Staubli VAL3: getJointData.pgx

public program getJointData(string x_sItem (dimensions=1), num x_nIndex (dimensions=1), joint& x_jJoint (dimensions=1), bool& x_bResult (dimensions=1))
  local num i
  local num l_nResult
  local string l_sSession
begin
  // get the joint data from the specific session...
  x_bResult=false
  call saveData:getSession(l_sSession)
  // get the colletion type...
  if sSession!=l_sSession
    // copy back
    sSession=l_sSession
    // load the actual one
    l_nResult=jt:libLoad(saveData:sPathTraj+"JPOINT")
    delay(0)
  endIf
  // use the type...
  if l_nResult==0 and isDefined(jt:tTraj[x_sItem]) and size(jt:tTraj[x_sItem].tData.jJoint)>x_nIndex
    // get the JOINT DATA
    x_jJoint=jt:tTraj[x_sItem].tData.jJoint[x_nIndex]
    delay(0)
    x_bResult=true
  endIf
end
